{attribute 'GeneratedUsingTerminal: EPP9022-0060-0017'}
{attribute addProperty BoxType "EPP9022-0060-0017"}
{attribute addProperty Id "StatusAT %I*Status_51F572C810VoltageAT %I*DINT4CurrentAT %I*DINT4"}
{attribute addProperty CRC "3106171789"}
{attribute addProperty Size "18"}
TYPE EPM_Inputs_Channel_B9246B8D :
STRUCT
	{attribute addProperty Name "Status"}
	Status AT %I* : Status_51F572C8;
	{attribute addProperty Name "Voltage"}
	Voltage AT %I* : DINT;
	{attribute addProperty Name "Current"}
	Current AT %I* : DINT;
END_STRUCT
END_TYPE

(* stored: Version 1.2.0.0, ProductVersion 3.1.4024.9
   DUT EPM_Inputs_Channel_B9246B8D: Id {68c2241a-c252-4481-9148-29d1a1c6cd98} *)
